Staubli VAL3: Main.dtx

bool bInputBuffering
bool bTaskManager
jointRx jHome
mdesc mNomSpeed
num nInputBuffer[136]
  [0] = 1
  [4] = 255
  [5] = 255
  [6] = 255
  [7] = 255
  [8] = 15
  [14] = 164
  [15] = 66
  [58] = 72
  [59] = 66
  [98] = 200
  [99] = 65
  [102] = 200
  [103] = 65
num nMessageBuffer[34 4]
  [0,0] = 1
  [1,0] = 255
  [1,1] = 255
  [1,2] = 255
  [1,3] = 255
  [2,0] = 15
  [3,2] = 164
  [3,3] = 66
  [14,2] = 72
  [14,3] = 66
  [24,2] = 200
  [24,3] = 65
  [25,2] = 200
  [25,3] = 65
sio siConn = {link=Socket\subscriber}
sio soConn = {link=Socket\publisher}
string sInputBuffering = "subscriber"
